{attribute 'linkalways'} 
{attribute 'no_explicit_call' := 'This FB is a CLASS and must be accessed using methods or properties'}
{attribute 'enable_dynamic_creation'}
FUNCTION_BLOCK INTERNAL DefaultMoveAbsoluteBuilder IMPLEMENTS MoveAbsoluteBuilder
VAR
	parent_builder : MotionBuilder;
	parameters : REFERENCE TO BuilderParameters;
END_VAR

METHOD PUBLIC Acceleration : MoveAbsoluteBuilder
VAR_INPUT
	value : LREAL;
END_VAR
parent_builder.Acceleration(value);
Acceleration := THIS^;
END_METHOD

METHOD PUBLIC BufferMode : MoveAbsoluteBuilder
VAR_INPUT
	mode : MotionBufferMode;
END_VAR
parent_builder.BufferMode(mode);
BufferMode := THIS^;
END_METHOD

METHOD PUBLIC BuildMoveAbsoluteCommand : MotionCommand
VAR_INPUT
	axis : REFERENCE TO Mc2Axis;
END_VAR
VAR
	command_ptr : POINTER TO MoveAbsoluteCommand;
	command : MotionCommand;
END_VAR
command_ptr := __NEW(MoveAbsoluteCommand(
	axis := axis,
	position := parameters.position,
	velocity := parameters.velocity,
	acceleration := parameters.acceleration,
	deceleration := parameters.deceleration,
	jerk := parameters.jerk,
	buffer_mode := parameters.buffer_mode
));
BuildMoveAbsoluteCommand := command_ptr^;
END_METHOD

METHOD PUBLIC Deceleration : MoveAbsoluteBuilder
VAR_INPUT
	value : LREAL;
END_VAR
parent_builder.Deceleration(value);
Deceleration := THIS^;
END_METHOD

//FB_Init is always available implicitly and it is used primarily for initialization.
//The return value is not evaluated. For a specific influence, you can also declare the
//methods explicitly and provide additional code there with the standard initialization
//code. You can evaluate the return value.
METHOD FB_Init: BOOL
VAR_INPUT
    bInitRetains : BOOL; // TRUE: the retain variables are initialized (reset warm / reset cold)
    bInCopyCode : BOOL;  // TRUE: the instance will be copied to the copy code afterward (online change)
	parent_builder : MotionBuilder;
	parameters : REFERENCE TO BuilderParameters;
END_VAR
THIS^.parent_builder := parent_builder;
THIS^.parameters REF= parameters;
END_METHOD

METHOD PUBLIC Jerk : MoveAbsoluteBuilder
VAR_INPUT
	value : LREAL;
END_VAR
parent_builder.Jerk(value);
Jerk := THIS^;
END_METHOD

METHOD PUBLIC Position : MoveAbsoluteBuilder
VAR_INPUT
	value : LREAL;
END_VAR
parent_builder.Position(value);
Position := THIS^;
END_METHOD

METHOD PUBLIC Reset : MoveAbsoluteBuilder
parent_builder.Reset();
Reset := THIS^;
END_METHOD

METHOD PUBLIC Velocity : MoveAbsoluteBuilder
VAR_INPUT
	value : LREAL;
END_VAR
parent_builder.Velocity(value);
Velocity := THIS^;
END_METHOD

END_FUNCTION_BLOCK

(* stored: Version 1.1.0.1
   POU DefaultMoveAbsoluteBuilder: Id {2200d402-ea56-0101-341c-600ac2ad507a}, SpecialFunc None
   Folder Builders: Id {ed6901ad-55a4-0f9f-1cb6-f0fdf076c8d9}
   Folder Constructor: Id {32574500-4dea-0e52-0ec8-c9fdc7cdcf03}
   Folder PropertySetters: Id {c5bddcb0-9e9a-0f6f-3867-17647dbb61ba}
   Method Acceleration: Id {c50a551d-b2b5-0f79-1863-ec2c8e4f587a}
   Method BufferMode: Id {94111ddf-7e48-0022-3e3f-858e7b61f5b8}
   Method BuildMoveAbsoluteCommand: Id {25567da8-96d8-0d92-11ec-c0615cca58cf}
   Method Deceleration: Id {142a90fc-c1e7-0a06-34b9-ffb1441370a1}
   Method FB_Init: Id {5edbc7f8-c8e4-0730-33be-76fb3b2f1dcc}
   Method Jerk: Id {925ebf38-d200-0d82-2f5f-d009e500eb67}
   Method Position: Id {b2cb9594-c116-0887-2b7c-7524b6fe02ed}
   Method Reset: Id {fff619f8-9807-03a6-38d0-3067a5993487}
   Method Velocity: Id {568c5770-128b-0124-2a8e-8b07c24536f2} *)
